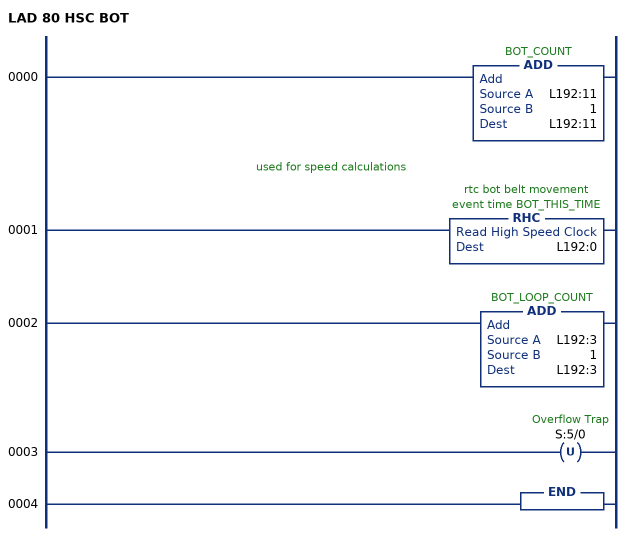
% Rung: 0 %
SOR ADD L192:11 1 L192:11 EOR
%   L192:11  BOT_COUNT %
% Rung: 1 %
% used for speed calculations %
SOR RHC L192:0 EOR
%   L192:0  BOT_THIS_TIME  "rtc bot belt movement event time" %
% Rung: 2 %
SOR ADD L192:3 1 L192:3 EOR
%   L192:3  BOT_LOOP_COUNT %
% Rung: 3 %
SOR OTU S:5/0 EOR
%   S:5/0  "Overflow Trap" %
% Rung: 4 %
SOR END EOR

LADDER 90 "HSC TOP"
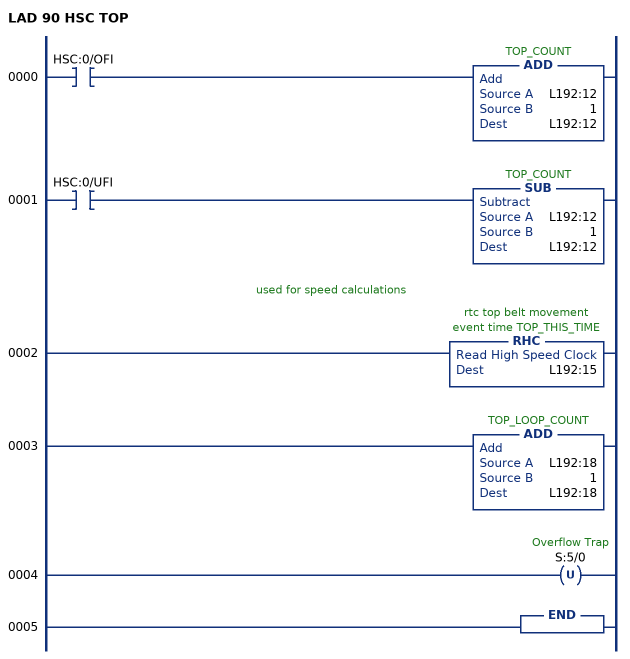
% Rung: 0 %
SOR XIC HSC:0/OFI ADD L192:12 1 L192:12 EOR
%   L192:12  TOP_COUNT %
% Rung: 1 %
SOR XIC HSC:0/UFI SUB L192:12 1 L192:12 EOR
%   L192:12  TOP_COUNT %
% Rung: 2 %
% used for speed calculations %
SOR RHC L192:15 EOR
%   L192:15  TOP_THIS_TIME  "rtc top belt movement event time" %
% Rung: 3 %
SOR ADD L192:18 1 L192:18 EOR
%   L192:18  TOP_LOOP_COUNT %
% Rung: 4 %
SOR OTU S:5/0 EOR
%   S:5/0  "Overflow Trap" %
% Rung: 5 %
SOR END EOR

LADDER 100 "1 MS STI"    % high speed %
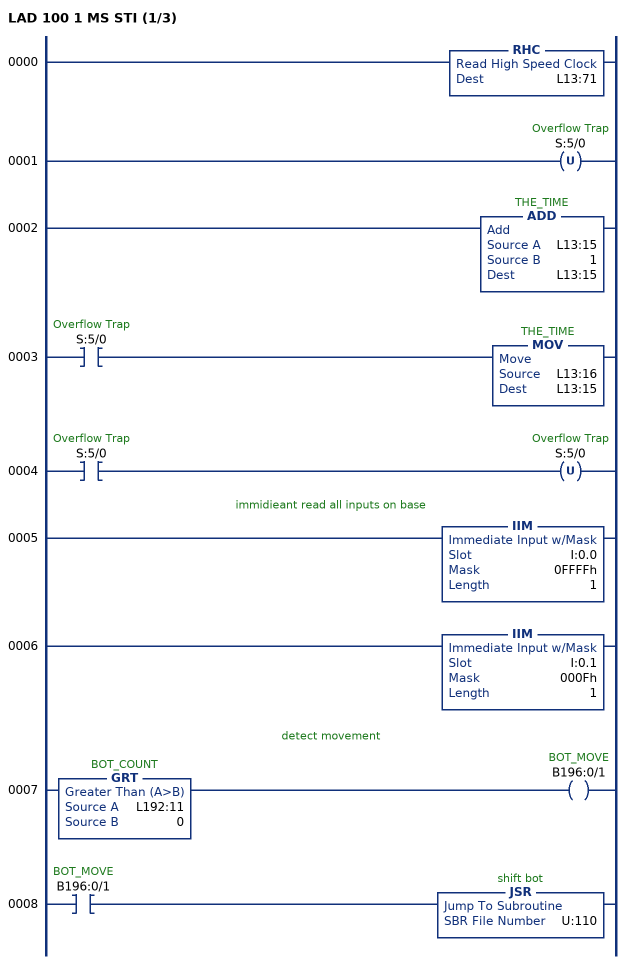
% Rung: 0 %
SOR RHC L13:71 EOR
% Rung: 1 %
SOR OTU S:5/0 EOR
%   S:5/0  "Overflow Trap" %
% Rung: 2 %
SOR ADD L13:15 1 L13:15 EOR
%   L13:15  THE_TIME %
% Rung: 3 %
SOR XIC S:5/0 MOV L13:16 L13:15 EOR
%   S:5/0  "Overflow Trap" %
%   L13:16  MIN_LONG %
%   L13:15  THE_TIME %
% Rung: 4 %
SOR XIC S:5/0 OTU S:5/0 EOR
%   S:5/0  "Overflow Trap" %
% Rung: 5 %
% immidieant read all inputs on base %
SOR IIM I:0.0 0FFFFh 1 EOR
% Rung: 6 %
SOR IIM I:0.1 000Fh 1 EOR
% Rung: 7 %
% detect movement %
SOR GRT L192:11 0 OTE B196:0/1 EOR
%   L192:11  BOT_COUNT %
%   B196:0/1  BOT_MOVE %
% Rung: 8 %
SOR XIC B196:0/1 JSR U:110 EOR
%   B196:0/1  BOT_MOVE %
%   U:110  "shift bot" %

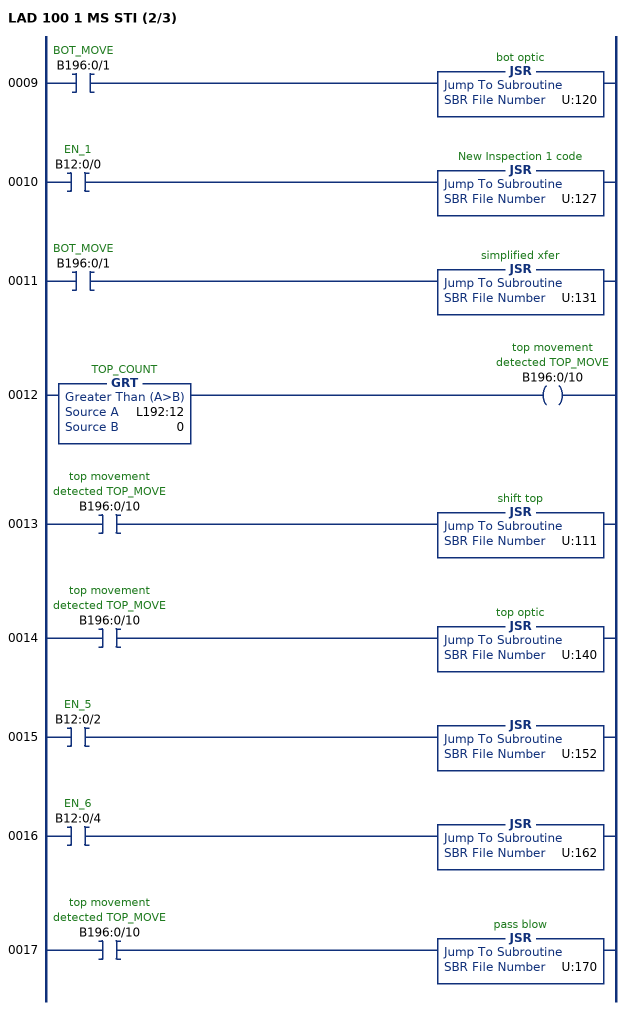
% Rung: 9 %
SOR XIC B196:0/1 JSR U:120 EOR
%   B196:0/1  BOT_MOVE %
%   U:120  "bot optic" %
% Rung: 10 %
SOR XIC B12:0/0 JSR U:127 EOR
%   B12:0/0  EN_1 %
%   U:127  "New Inspection 1 code" %
% Rung: 11 %
SOR XIC B196:0/1 JSR U:131 EOR
%   B196:0/1  BOT_MOVE %
%   U:131  "simplified xfer" %
% Rung: 12 %
SOR GRT L192:12 0 OTE B196:0/10 EOR
%   L192:12  TOP_COUNT %
%   B196:0/10  TOP_MOVE  "top movement detected" %
% Rung: 13 %
SOR XIC B196:0/10 JSR U:111 EOR
%   B196:0/10  TOP_MOVE  "top movement detected" %
%   U:111  "shift top" %
% Rung: 14 %
SOR XIC B196:0/10 JSR U:140 EOR
%   B196:0/10  TOP_MOVE  "top movement detected" %
%   U:140  "top optic" %
% Rung: 15 %
SOR XIC B12:0/2 JSR U:152 EOR
%   B12:0/2  EN_5 %
% Rung: 16 %
SOR XIC B12:0/4 JSR U:162 EOR
%   B12:0/4  EN_6 %
% Rung: 17 %
SOR XIC B196:0/10 JSR U:170 EOR
%   B196:0/10  TOP_MOVE  "top movement detected" %
%   U:170  "pass blow" %

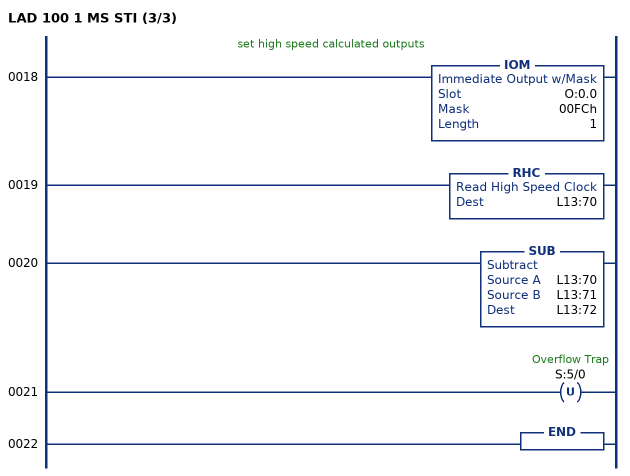
% Rung: 18 %
% set high speed calculated outputs %
SOR IOM O:0.0 00FCh 1 EOR
% Rung: 19 %
SOR RHC L13:70 EOR
% Rung: 20 %
SOR SUB L13:70 L13:71 L13:72 EOR
% Rung: 21 %
SOR OTU S:5/0 EOR
%   S:5/0  "Overflow Trap" %
% Rung: 22 %
SOR END EOR

LADDER 102 "SPEED BOT"    % high speed %
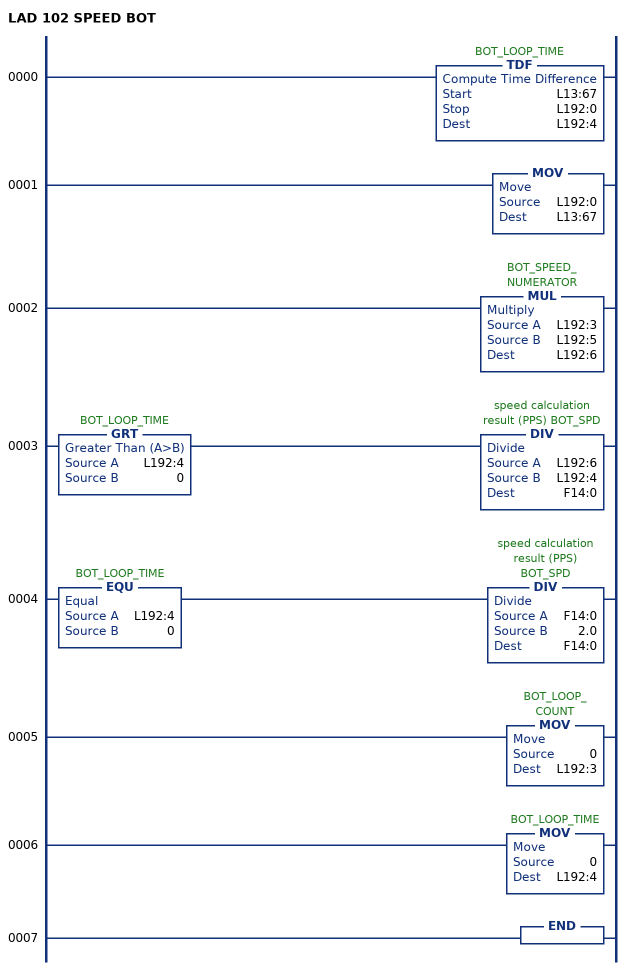
% Rung: 0 %
SOR TDF L13:67 L192:0 L192:4 EOR
%   L192:0  BOT_THIS_TIME  "rtc bot belt movement event time" %
%   L192:4  BOT_LOOP_TIME %
% Rung: 1 %
SOR MOV L192:0 L13:67 EOR
%   L192:0  BOT_THIS_TIME  "rtc bot belt movement event time" %
% Rung: 2 %
SOR MUL L192:3 L192:5 L192:6 EOR
%   L192:3  BOT_LOOP_COUNT %
%   L192:5  TKS_PER_SECOND %
%   L192:6  BOT_SPEED_NUMERATOR %
% Rung: 3 %
SOR GRT L192:4 0 DIV L192:6 L192:4 F14:0 EOR
%   L192:4  BOT_LOOP_TIME %
%   L192:6  BOT_SPEED_NUMERATOR %
%   F14:0  BOT_SPD  "speed calculation result (PPS)" %
% Rung: 4 %
SOR EQU L192:4 0 DIV F14:0 2.0 F14:0 EOR
%   L192:4  BOT_LOOP_TIME %
%   F14:0  BOT_SPD  "speed calculation result (PPS)" %
% Rung: 5 %
SOR MOV 0 L192:3 EOR
%   L192:3  BOT_LOOP_COUNT %
% Rung: 6 %
SOR MOV 0 L192:4 EOR
%   L192:4  BOT_LOOP_TIME %
% Rung: 7 %
SOR END EOR

LADDER 103 "SPEED TOP"    % high speed %
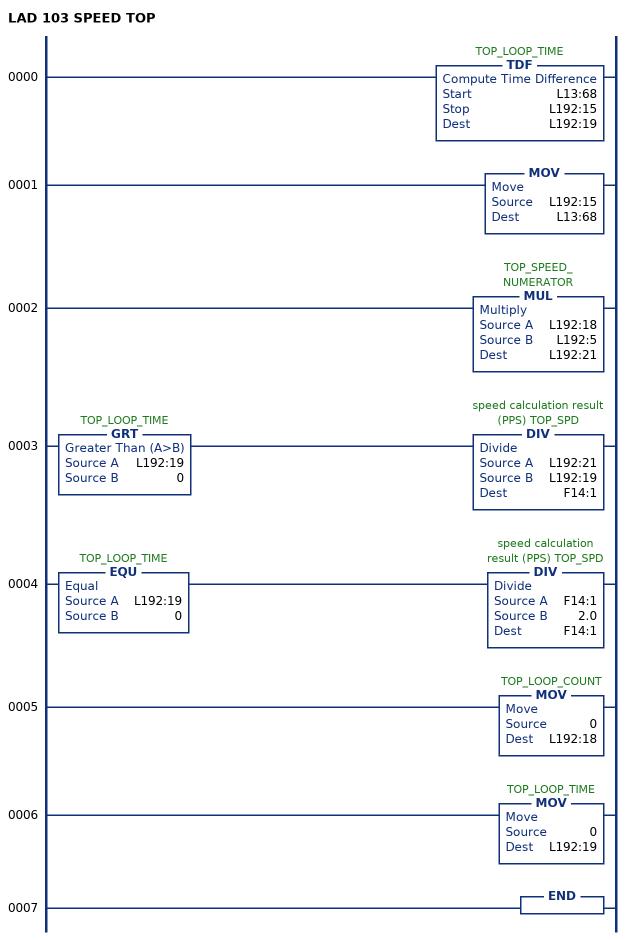
% Rung: 0 %
SOR TDF L13:68 L192:15 L192:19 EOR
%   L192:15  TOP_THIS_TIME  "rtc top belt movement event time" %
%   L192:19  TOP_LOOP_TIME %
% Rung: 1 %
SOR MOV L192:15 L13:68 EOR
%   L192:15  TOP_THIS_TIME  "rtc top belt movement event time" %
% Rung: 2 %
SOR MUL L192:18 L192:5 L192:21 EOR
%   L192:18  TOP_LOOP_COUNT %
%   L192:5  TKS_PER_SECOND %
%   L192:21  TOP_SPEED_NUMERATOR %
% Rung: 3 %
SOR GRT L192:19 0 DIV L192:21 L192:19 F14:1 EOR
%   L192:19  TOP_LOOP_TIME %
%   L192:21  TOP_SPEED_NUMERATOR %
%   F14:1  TOP_SPD  "speed calculation result (PPS)" %
% Rung: 4 %
SOR EQU L192:19 0 DIV F14:1 2.0 F14:1 EOR
%   L192:19  TOP_LOOP_TIME %
%   F14:1  TOP_SPD  "speed calculation result (PPS)" %
% Rung: 5 %
SOR MOV 0 L192:18 EOR
%   L192:18  TOP_LOOP_COUNT %
% Rung: 6 %
SOR MOV 0 L192:19 EOR
%   L192:19  TOP_LOOP_TIME %
% Rung: 7 %
SOR END EOR

LADDER 104 "P BOT"    % high speed %
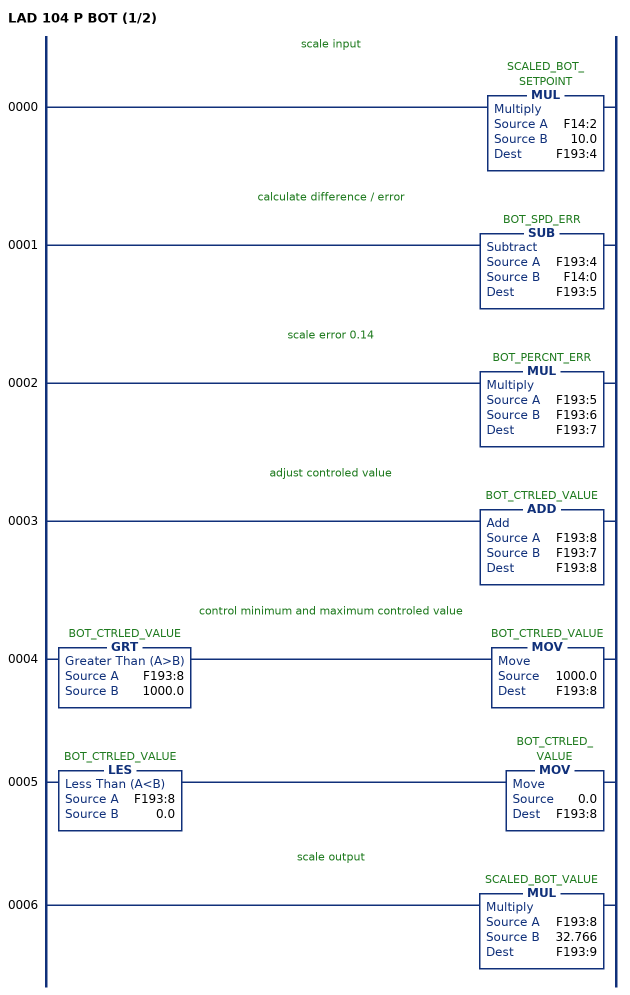
% Rung: 0 %
% scale input %
SOR MUL F14:2 10.0 F193:4 EOR
%   F14:2  BOT_SPD_SETPOINT %
%   F193:4  SCALED_BOT_SETPOINT %
% Rung: 1 %
% calculate difference / error %
SOR SUB F193:4 F14:0 F193:5 EOR
%   F193:4  SCALED_BOT_SETPOINT %
%   F14:0  BOT_SPD  "speed calculation result (PPS)" %
%   F193:5  BOT_SPD_ERR %
% Rung: 2 %
% scale error 0.14 %
SOR MUL F193:5 F193:6 F193:7 EOR
%   F193:5  BOT_SPD_ERR %
%   F193:6  BOT_FDBK_RATIO %
%   F193:7  BOT_PERCNT_ERR %
% Rung: 3 %
% adjust controled value %
SOR ADD F193:8 F193:7 F193:8 EOR
%   F193:8  BOT_CTRLED_VALUE %
%   F193:7  BOT_PERCNT_ERR %
% Rung: 4 %
% control minimum and maximum controled value %
SOR GRT F193:8 1000.0 MOV 1000.0 F193:8 EOR
%   F193:8  BOT_CTRLED_VALUE %
% Rung: 5 %
SOR LES F193:8 0.0 MOV 0.0 F193:8 EOR
%   F193:8  BOT_CTRLED_VALUE %
% Rung: 6 %
% scale output %
SOR MUL F193:8 32.766 F193:9 EOR
%   F193:8  BOT_CTRLED_VALUE %
%   F193:9  SCALED_BOT_VALUE %

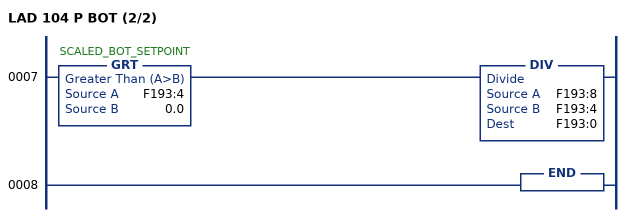
% Rung: 7 %
SOR GRT F193:4 0.0 DIV F193:8 F193:4 F193:0 EOR
%   F193:4  SCALED_BOT_SETPOINT %
%   F193:8  BOT_CTRLED_VALUE %
% Rung: 8 %
SOR END EOR

LADDER 105 "P TOP"    % high speed %
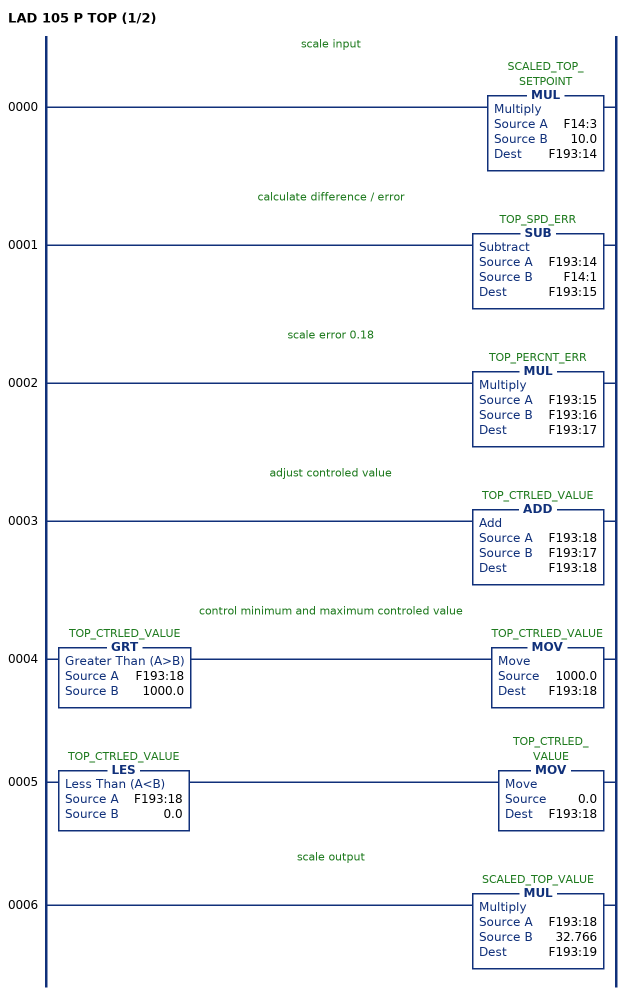
% Rung: 0 %
% scale input %
SOR MUL F14:3 10.0 F193:14 EOR
%   F14:3  TOP_SPD_SETPOINT %
%   F193:14  SCALED_TOP_SETPOINT %
% Rung: 1 %
% calculate difference / error %
SOR SUB F193:14 F14:1 F193:15 EOR
%   F193:14  SCALED_TOP_SETPOINT %
%   F14:1  TOP_SPD  "speed calculation result (PPS)" %
%   F193:15  TOP_SPD_ERR %
% Rung: 2 %
% scale error 0.18 %
SOR MUL F193:15 F193:16 F193:17 EOR
%   F193:15  TOP_SPD_ERR %
%   F193:16  TOP_FDBK_RATIO %
%   F193:17  TOP_PERCNT_ERR %
% Rung: 3 %
% adjust controled value %
SOR ADD F193:18 F193:17 F193:18 EOR
%   F193:18  TOP_CTRLED_VALUE %
%   F193:17  TOP_PERCNT_ERR %
% Rung: 4 %
% control minimum and maximum controled value %
SOR GRT F193:18 1000.0 MOV 1000.0 F193:18 EOR
%   F193:18  TOP_CTRLED_VALUE %
% Rung: 5 %
SOR LES F193:18 0.0 MOV 0.0 F193:18 EOR
%   F193:18  TOP_CTRLED_VALUE %
% Rung: 6 %
% scale output %
SOR MUL F193:18 32.766 F193:19 EOR
%   F193:18  TOP_CTRLED_VALUE %
%   F193:19  SCALED_TOP_VALUE %

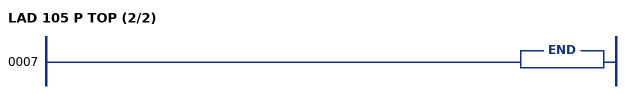
% Rung: 7 %
SOR END EOR

LADDER 110 "SHIFT BOT"
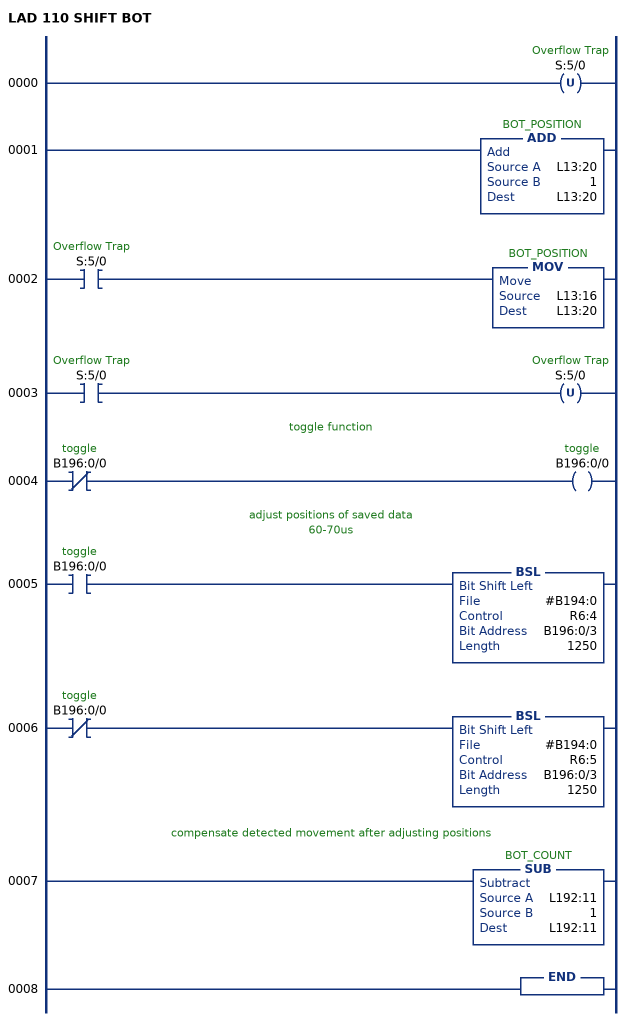
% Rung: 0 %
SOR OTU S:5/0 EOR
%   S:5/0  "Overflow Trap" %
% Rung: 1 %
SOR ADD L13:20 1 L13:20 EOR
%   L13:20  BOT_POSITION %
% Rung: 2 %
SOR XIC S:5/0 MOV L13:16 L13:20 EOR
%   S:5/0  "Overflow Trap" %
%   L13:16  MIN_LONG %
%   L13:20  BOT_POSITION %
% Rung: 3 %
SOR XIC S:5/0 OTU S:5/0 EOR
%   S:5/0  "Overflow Trap" %
% Rung: 4 %
% toggle function %
SOR XIO B196:0/0 OTE B196:0/0 EOR
%   B196:0/0  "toggle" %
% Rung: 5 %
% adjust positions of saved data
% 60-70us %
SOR XIC B196:0/0 BSL #B194:0 R6:4 B196:0/3 1250 EOR
%   B196:0/0  "toggle" %
%   B196:0/3  OFF %
% Rung: 6 %
SOR XIO B196:0/0 BSL #B194:0 R6:5 B196:0/3 1250 EOR
%   B196:0/0  "toggle" %
%   B196:0/3  OFF %
% Rung: 7 %
% compensate detected movement after adjusting positions %
SOR SUB L192:11 1 L192:11 EOR
%   L192:11  BOT_COUNT %
% Rung: 8 %
SOR END EOR

LADDER 111 "SHIFT TOP"
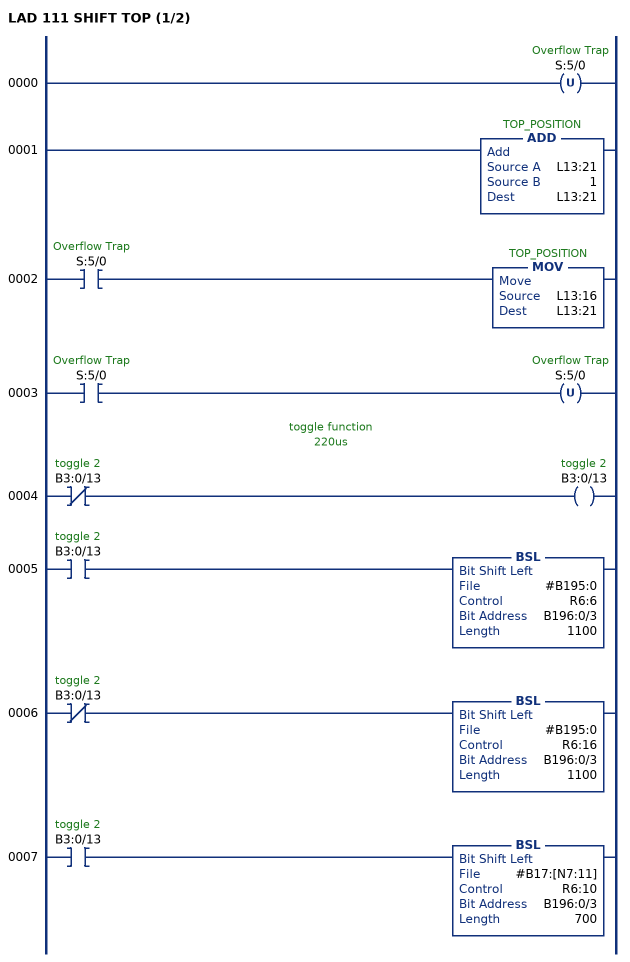
% Rung: 0 %
SOR OTU S:5/0 EOR
%   S:5/0  "Overflow Trap" %
% Rung: 1 %
SOR ADD L13:21 1 L13:21 EOR
%   L13:21  TOP_POSITION %
% Rung: 2 %
SOR XIC S:5/0 MOV L13:16 L13:21 EOR
%   S:5/0  "Overflow Trap" %
%   L13:16  MIN_LONG %
%   L13:21  TOP_POSITION %
% Rung: 3 %
SOR XIC S:5/0 OTU S:5/0 EOR
%   S:5/0  "Overflow Trap" %
% Rung: 4 %
% toggle function
% 220us %
SOR XIO B3:0/13 OTE B3:0/13 EOR
%   B3:0/13  "toggle 2" %
% Rung: 5 %
SOR XIC B3:0/13 BSL #B195:0 R6:6 B196:0/3 1100 EOR
%   B3:0/13  "toggle 2" %
%   R6:6  "from top load to top optic" %
%   B196:0/3  OFF %
% Rung: 6 %
SOR XIO B3:0/13 BSL #B195:0 R6:16 B196:0/3 1100 EOR
%   B3:0/13  "toggle 2" %
%   B196:0/3  OFF %
% Rung: 7 %
SOR XIC B3:0/13 BSL #B17:[N7:11] R6:10 B196:0/3 700 EOR
%   B3:0/13  "toggle 2" %
%   B196:0/3  OFF %

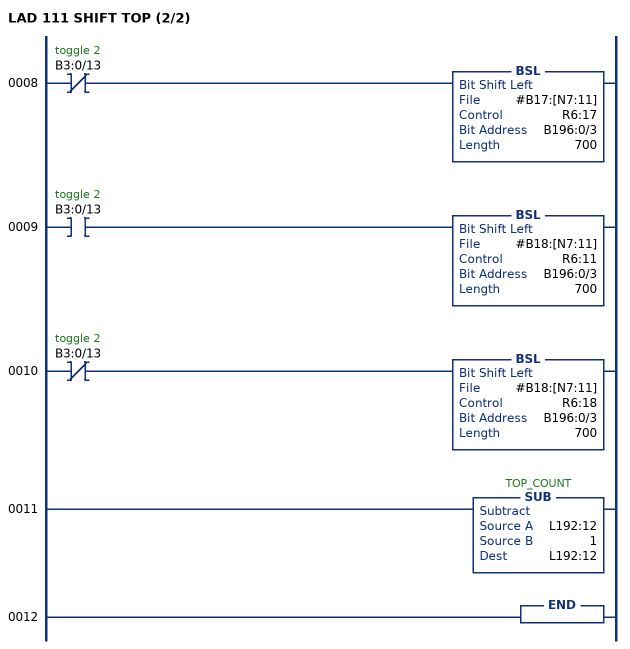
% Rung: 8 %
SOR XIO B3:0/13 BSL #B17:[N7:11] R6:17 B196:0/3 700 EOR
%   B3:0/13  "toggle 2" %
%   B196:0/3  OFF %
% Rung: 9 %
SOR XIC B3:0/13 BSL #B18:[N7:11] R6:11 B196:0/3 700 EOR
%   B3:0/13  "toggle 2" %
%   B196:0/3  OFF %
% Rung: 10 %
SOR XIO B3:0/13 BSL #B18:[N7:11] R6:18 B196:0/3 700 EOR
%   B3:0/13  "toggle 2" %
%   B196:0/3  OFF %
% Rung: 11 %
SOR SUB L192:12 1 L192:12 EOR
%   L192:12  TOP_COUNT %
% Rung: 12 %
SOR END EOR

LADDER 120 "BOTOPTIC"
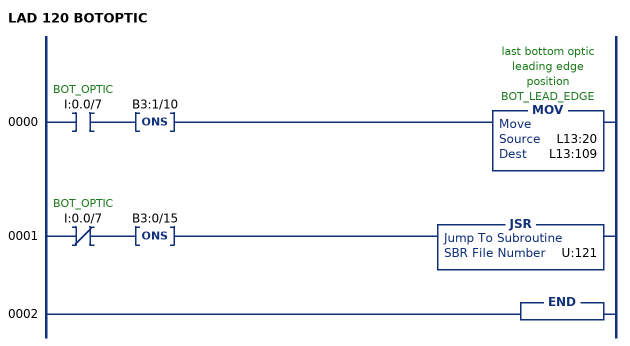
% Rung: 0 %
SOR XIC I:0.0/7 ONS B3:1/10 MOV L13:20 L13:109 EOR
%   I:0.0/7  BOT_OPTIC %
%   L13:20  BOT_POSITION %
%   L13:109  BOT_LEAD_EDGE  "last bottom optic leading edge position" %
% Rung: 1 %
SOR XIO I:0.0/7 ONS B3:0/15 JSR U:121 EOR
%   I:0.0/7  BOT_OPTIC %
% Rung: 2 %
SOR END EOR

LADDER 121 "BOTOPTMES"
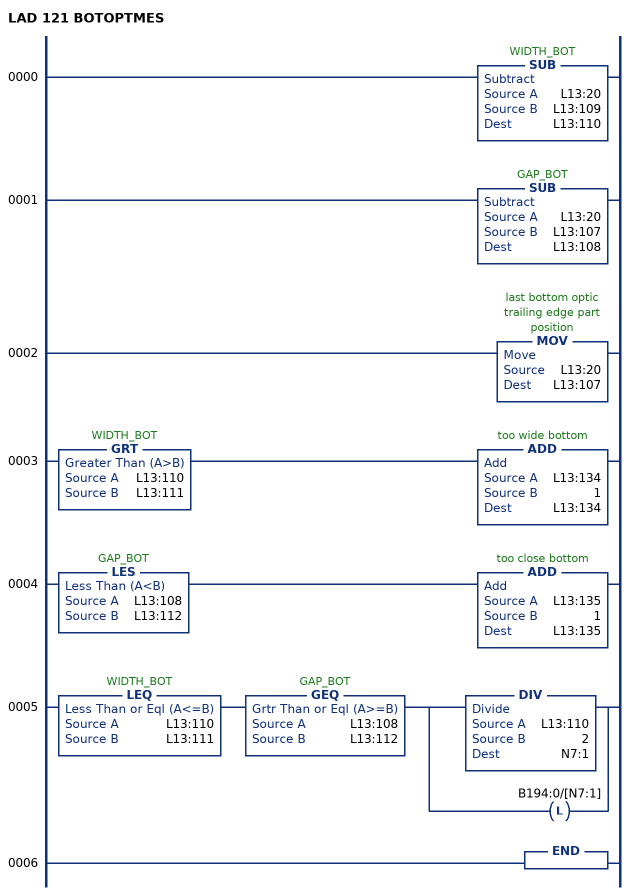
% Rung: 0 %
SOR SUB L13:20 L13:109 L13:110 EOR
%   L13:20  BOT_POSITION %
%   L13:109  BOT_LEAD_EDGE  "last bottom optic leading edge position" %
%   L13:110  WIDTH_BOT %
% Rung: 1 %
SOR SUB L13:20 L13:107 L13:108 EOR
%   L13:20  BOT_POSITION %
%   L13:107  "last bottom optic trailing edge part position" %
%   L13:108  GAP_BOT %
% Rung: 2 %
SOR MOV L13:20 L13:107 EOR
%   L13:20  BOT_POSITION %
%   L13:107  "last bottom optic trailing edge part position" %
% Rung: 3 %
SOR GRT L13:110 L13:111 ADD L13:134 1 L13:134 EOR
%   L13:110  WIDTH_BOT %
%   L13:111  BOT_MAX_WIDTH %
%   L13:134  "too wide bottom" %
% Rung: 4 %
SOR LES L13:108 L13:112 ADD L13:135 1 L13:135 EOR
%   L13:108  GAP_BOT %
%   L13:112  BOT_MIN_GAP %
%   L13:135  "too close bottom" %
% Rung: 5 %
SOR LEQ L13:110 L13:111 GEQ L13:108 L13:112 BST DIV L13:110 2 N7:1 NXB OTL B194:0/[N7:1] BND EOR
%   L13:110  WIDTH_BOT %
%   L13:111  BOT_MAX_WIDTH %
%   L13:108  GAP_BOT %
%   L13:112  BOT_MIN_GAP %
% Rung: 6 %
SOR END EOR

LADDER 124 "INS1RESULT"
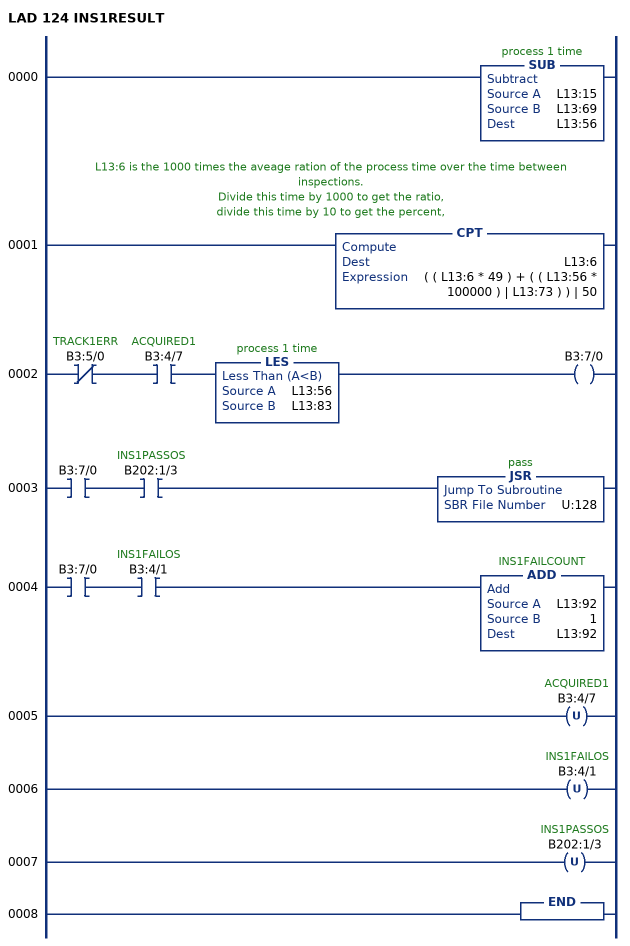
% Rung: 0 %
SOR SUB L13:15 L13:69 L13:56 EOR
%   L13:15  THE_TIME %
%   L13:69  TIMEOFACQ1  "the time of the last acquire" %
%   L13:56  "process 1 time" %
% Rung: 1 %
% L13:6 is the 1000 times the aveage ration of the process time over the time between inspections.
% Divide this time by 1000 to get the ratio,
% divide this time by 10 to get the percent, %
SOR CPT L13:6 " ( ( L13:6 * 49 ) + ( ( L13:56 * 100000 ) | L13:73 ) ) | 50 " EOR
%   L13:56  "process 1 time" %
%   L13:73  TBI %
% Rung: 2 %
SOR XIO B3:5/0 XIC B3:4/7 LES L13:56 L13:83 OTE B3:7/0 EOR
%   B3:5/0  TRACK1ERR %
%   B3:4/7  ACQUIRED1 %
%   L13:56  "process 1 time" %
% Rung: 3 %
SOR XIC B3:7/0 XIC B202:1/3 JSR U:128 EOR
%   B202:1/3  INS1PASSOS %
%   U:128  "pass" %
% Rung: 4 %
SOR XIC B3:7/0 XIC B3:4/1 ADD L13:92 1 L13:92 EOR
%   B3:4/1  INS1FAILOS %
%   L13:92  INS1FAILCOUNT %
% Rung: 5 %
SOR OTU B3:4/7 EOR
%   B3:4/7  ACQUIRED1 %
% Rung: 6 %
SOR OTU B3:4/1 EOR
%   B3:4/1  INS1FAILOS %
% Rung: 7 %
SOR OTU B202:1/3 EOR
%   B202:1/3  INS1PASSOS %
% Rung: 8 %
SOR END EOR

LADDER 125 "FIXERR1"
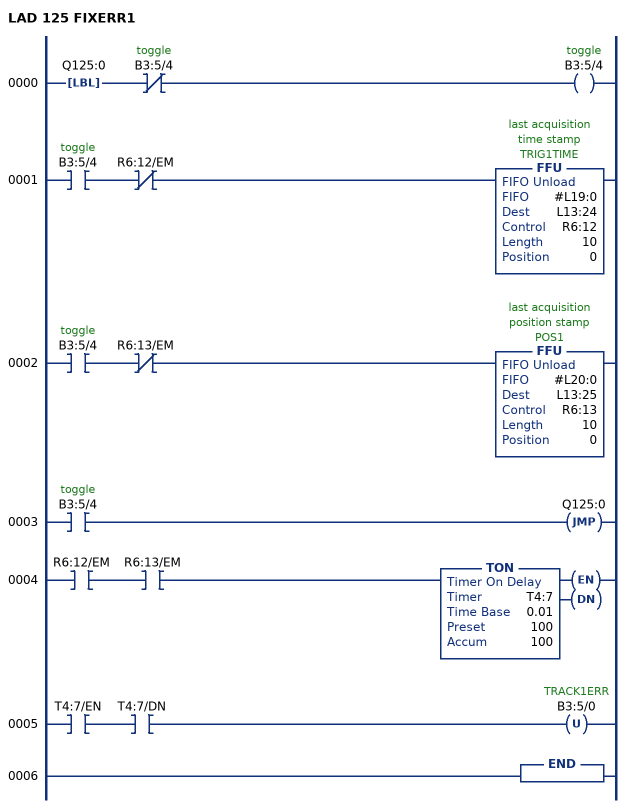
% Rung: 0 %
SOR LBL Q125:0 XIO B3:5/4 OTE B3:5/4 EOR
%   B3:5/4  "toggle" %
% Rung: 1 %
SOR XIC B3:5/4 XIO R6:12/EM FFU #L19:0 L13:24 R6:12 10 0 EOR
%   B3:5/4  "toggle" %
%   L13:24  TRIG1TIME  "last acquisition time stamp" %
% Rung: 2 %
SOR XIC B3:5/4 XIO R6:13/EM FFU #L20:0 L13:25 R6:13 10 0 EOR
%   B3:5/4  "toggle" %
%   L13:25  POS1  "last acquisition position stamp" %
% Rung: 3 %
SOR XIC B3:5/4 JMP Q125:0 EOR
%   B3:5/4  "toggle" %
% Rung: 4 %
SOR XIC R6:12/EM XIC R6:13/EM TON T4:7 0.01 100 100 EOR
% Rung: 5 %
SOR XIC T4:7/EN XIC T4:7/DN OTU B3:5/0 EOR
%   B3:5/0  TRACK1ERR %
% Rung: 6 %
SOR END EOR

LADDER 127 "INS1"
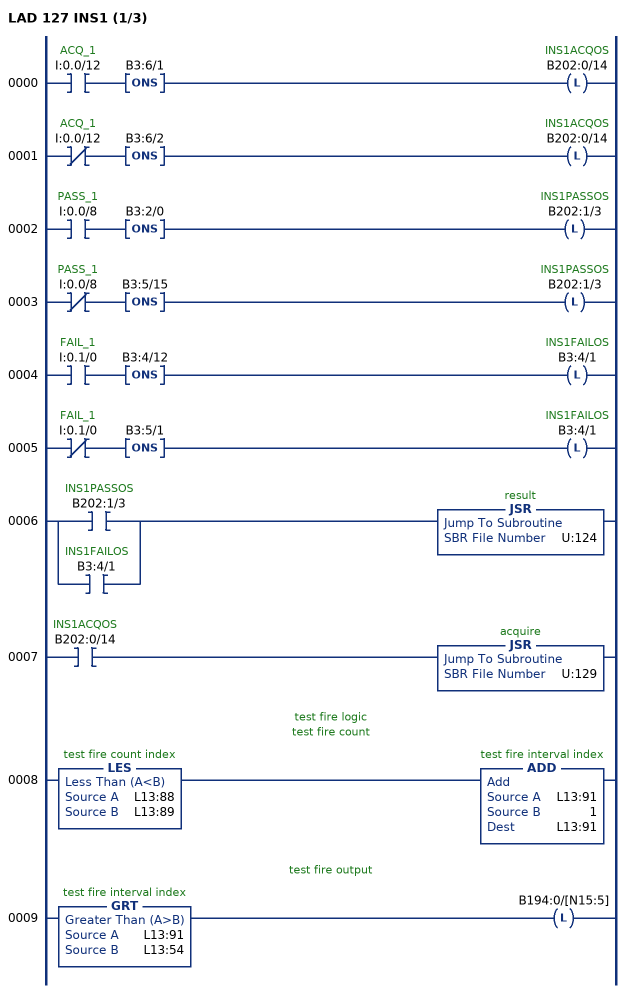
% Rung: 0 %
SOR XIC I:0.0/12 ONS B3:6/1 OTL B202:0/14 EOR
%   I:0.0/12  ACQ_1 %
%   B202:0/14  INS1ACQOS %
% Rung: 1 %
SOR XIO I:0.0/12 ONS B3:6/2 OTL B202:0/14 EOR
%   I:0.0/12  ACQ_1 %
%   B202:0/14  INS1ACQOS %
% Rung: 2 %
SOR XIC I:0.0/8 ONS B3:2/0 OTL B202:1/3 EOR
%   I:0.0/8  PASS_1 %
%   B202:1/3  INS1PASSOS %
% Rung: 3 %
SOR XIO I:0.0/8 ONS B3:5/15 OTL B202:1/3 EOR
%   I:0.0/8  PASS_1 %
%   B202:1/3  INS1PASSOS %
% Rung: 4 %
SOR XIC I:0.1/0 ONS B3:4/12 OTL B3:4/1 EOR
%   I:0.1/0  FAIL_1 %
%   B3:4/1  INS1FAILOS %
% Rung: 5 %
SOR XIO I:0.1/0 ONS B3:5/1 OTL B3:4/1 EOR
%   I:0.1/0  FAIL_1 %
%   B3:4/1  INS1FAILOS %
% Rung: 6 %
SOR BST XIC B202:1/3 NXB XIC B3:4/1 BND JSR U:124 EOR
%   B202:1/3  INS1PASSOS %
%   B3:4/1  INS1FAILOS %
%   U:124  "result" %
% Rung: 7 %
SOR XIC B202:0/14 JSR U:129 EOR
%   B202:0/14  INS1ACQOS %
%   U:129  "acquire" %
% Rung: 8 %
% test fire logic
% 
% test fire count %
SOR LES L13:88 L13:89 ADD L13:91 1 L13:91 EOR
%   L13:88  "test fire count index" %
%   L13:89  "test fire count" %
%   L13:91  "test fire interval index" %
% Rung: 9 %
% test fire output %
SOR GRT L13:91 L13:54 OTL B194:0/[N15:5] EOR
%   L13:91  "test fire interval index" %
%   L13:54  "test fire interval" %
%   N15:5  INS_1_TRIG_LOC %

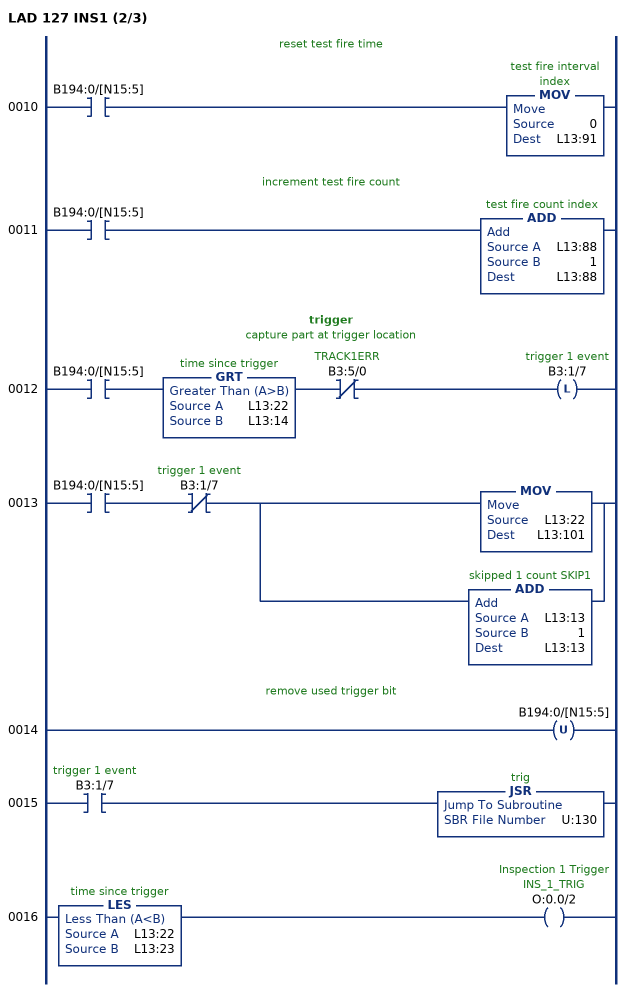
% Rung: 10 %
% reset test fire time %
SOR XIC B194:0/[N15:5] MOV 0 L13:91 EOR
%   N15:5  INS_1_TRIG_LOC %
%   L13:91  "test fire interval index" %
% Rung: 11 %
% increment test fire count %
SOR XIC B194:0/[N15:5] ADD L13:88 1 L13:88 EOR
%   N15:5  INS_1_TRIG_LOC %
%   L13:88  "test fire count index" %
% Rung: 12 %
% TITLE: trigger %
% capture part at trigger location %
SOR XIC B194:0/[N15:5] GRT L13:22 L13:14 XIO B3:5/0 OTL B3:1/7 EOR
%   N15:5  INS_1_TRIG_LOC %
%   L13:22  "time since trigger" %
%   B3:5/0  TRACK1ERR %
%   B3:1/7  "trigger 1 event" %
% Rung: 13 %
SOR XIC B194:0/[N15:5] XIO B3:1/7 BST MOV L13:22 L13:101 NXB ADD L13:13 1 L13:13 BND EOR
%   N15:5  INS_1_TRIG_LOC %
%   B3:1/7  "trigger 1 event" %
%   L13:22  "time since trigger" %
%   L13:13  SKIP1  "skipped 1 count" %
% Rung: 14 %
% remove used trigger bit %
SOR OTU B194:0/[N15:5] EOR
%   N15:5  INS_1_TRIG_LOC %
% Rung: 15 %
SOR XIC B3:1/7 JSR U:130 EOR
%   B3:1/7  "trigger 1 event" %
%   U:130  "trig" %
% Rung: 16 %
SOR LES L13:22 L13:23 OTE O:0.0/2 EOR
%   L13:22  "time since trigger" %
%   L13:23  "trigger on time" %
%   O:0.0/2  INS_1_TRIG  "Inspection 1 Trigger" %

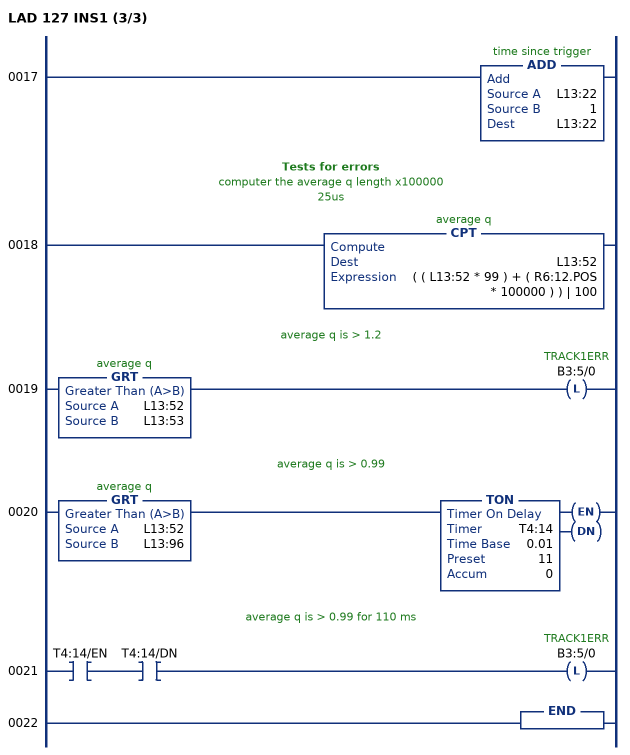
% Rung: 17 %
SOR ADD L13:22 1 L13:22 EOR
%   L13:22  "time since trigger" %
% Rung: 18 %
% TITLE: Tests for errors %
% computer the average q length x100000
% 25us %
SOR CPT L13:52 " ( ( L13:52 * 99 ) + ( R6:12.POS * 100000 ) ) | 100 " EOR
%   L13:52  "average q" %
% Rung: 19 %
% average q is > 1.2 %
SOR GRT L13:52 L13:53 OTL B3:5/0 EOR
%   L13:52  "average q" %
%   B3:5/0  TRACK1ERR %
% Rung: 20 %
% average q is > 0.99 %
SOR GRT L13:52 L13:96 TON T4:14 0.01 11 0 EOR
%   L13:52  "average q" %
% Rung: 21 %
% average q is > 0.99 for 110 ms %
SOR XIC T4:14/EN XIC T4:14/DN OTL B3:5/0 EOR
%   B3:5/0  TRACK1ERR %
% Rung: 22 %
SOR END EOR

LADDER 128 "INS1PASS"
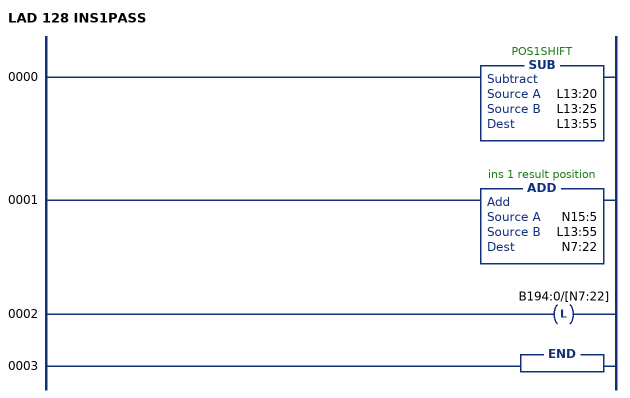
% Rung: 0 %
SOR SUB L13:20 L13:25 L13:55 EOR
%   L13:20  BOT_POSITION %
%   L13:25  POS1  "last acquisition position stamp" %
%   L13:55  POS1SHIFT %
% Rung: 1 %
SOR ADD N15:5 L13:55 N7:22 EOR
%   N15:5  INS_1_TRIG_LOC %
%   L13:55  POS1SHIFT %
%   N7:22  "ins 1 result position" %
% Rung: 2 %
SOR OTL B194:0/[N7:22] EOR
%   N7:22  "ins 1 result position" %
% Rung: 3 %
SOR END EOR

LADDER 129 "INS1ACQ"
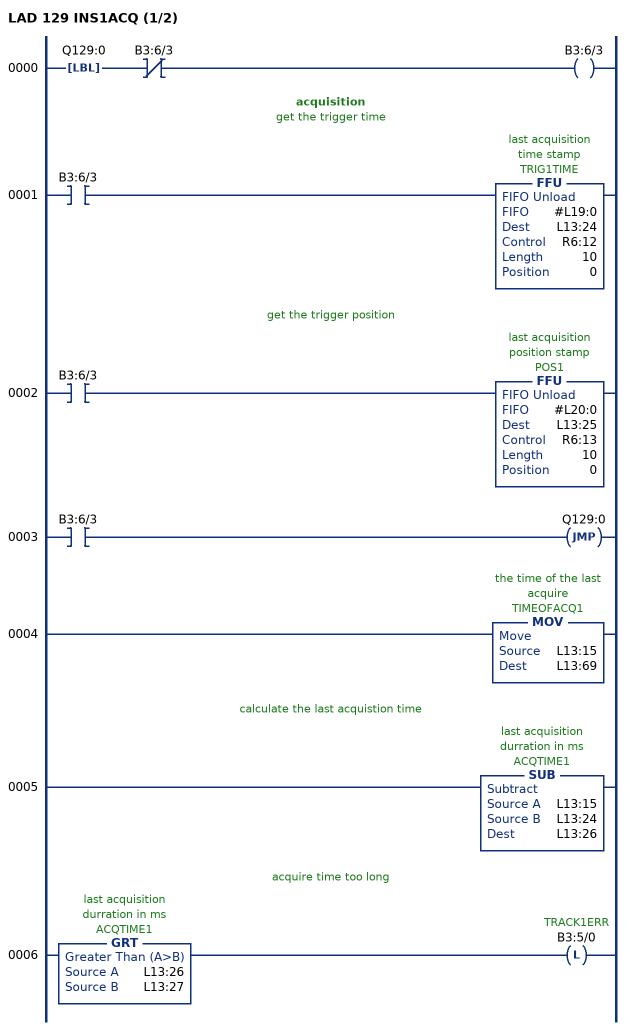
% Rung: 0 %
SOR LBL Q129:0 XIO B3:6/3 OTE B3:6/3 EOR
% Rung: 1 %
% TITLE: acquisition %
% get the trigger time %
SOR XIC B3:6/3 FFU #L19:0 L13:24 R6:12 10 0 EOR
%   L13:24  TRIG1TIME  "last acquisition time stamp" %
% Rung: 2 %
% get the trigger position %
SOR XIC B3:6/3 FFU #L20:0 L13:25 R6:13 10 0 EOR
%   L13:25  POS1  "last acquisition position stamp" %
% Rung: 3 %
SOR XIC B3:6/3 JMP Q129:0 EOR
% Rung: 4 %
SOR MOV L13:15 L13:69 EOR
%   L13:15  THE_TIME %
%   L13:69  TIMEOFACQ1  "the time of the last acquire" %
% Rung: 5 %
% calculate the last acquistion time %
SOR SUB L13:15 L13:24 L13:26 EOR
%   L13:15  THE_TIME %
%   L13:24  TRIG1TIME  "last acquisition time stamp" %
%   L13:26  ACQTIME1  "last acquisition durration in ms" %
% Rung: 6 %
% acquire time too long %
SOR GRT L13:26 L13:27 OTL B3:5/0 EOR
%   L13:26  ACQTIME1  "last acquisition durration in ms" %
%   L13:27  "max acquisition time in ms" %
%   B3:5/0  TRACK1ERR %

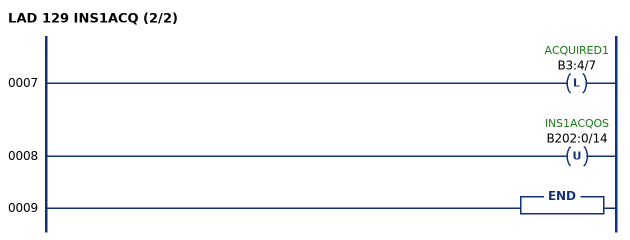
% Rung: 7 %
SOR OTL B3:4/7 EOR
%   B3:4/7  ACQUIRED1 %
% Rung: 8 %
SOR OTU B202:0/14 EOR
%   B202:0/14  INS1ACQOS %
% Rung: 9 %
SOR END EOR

LADDER 130 "INS1TRIG"
